{attribute 'GeneratedUsingTerminal: AES-D-BC-ECAT-0000'}
{attribute addProperty BoxType "AES-D-BC-ECAT-0000"}
{attribute addProperty Id "Switch_Count_StoreAT %Q*BOOL1HL_SwapAT %Q*BOOL1Default_Modul_ControlAT %Q*BOOL1"}
{attribute addProperty CRC "1482153743"}
{attribute addProperty Size "3"}
TYPE Device_Control_5857DF0F EXTENDS TcoIo.OutputBase_10CEE7DE :
STRUCT
	{attribute addProperty Name "Switch_Count_Store"}
	Switch_Count_Store AT %Q* : BOOL;
	{attribute addProperty Name "HL_Swap"}
	HL_Swap AT %Q* : BOOL;
	{attribute addProperty Name "Default_Modul_Control"}
	Default_Modul_Control AT %Q* : BOOL;
END_STRUCT
END_TYPE

(* stored: Version 1.2.0.0, ProductVersion 3.1.4024.11
   DUT Device_Control_5857DF0F: Id {943bc6bb-6ba5-043e-2d13-a69aae2e1db3} *)
